PROGRAM A25

END_PROGRAM

(* stored: Version 1.1.0.1, ProductVersion 3.1.4024.11
   POU A25: Id {3b04d2e6-0b6c-4c36-b7dd-d9e45e2be25d}, SpecialFunc None *)
